Universal Robots PolyScope program: programa.urp

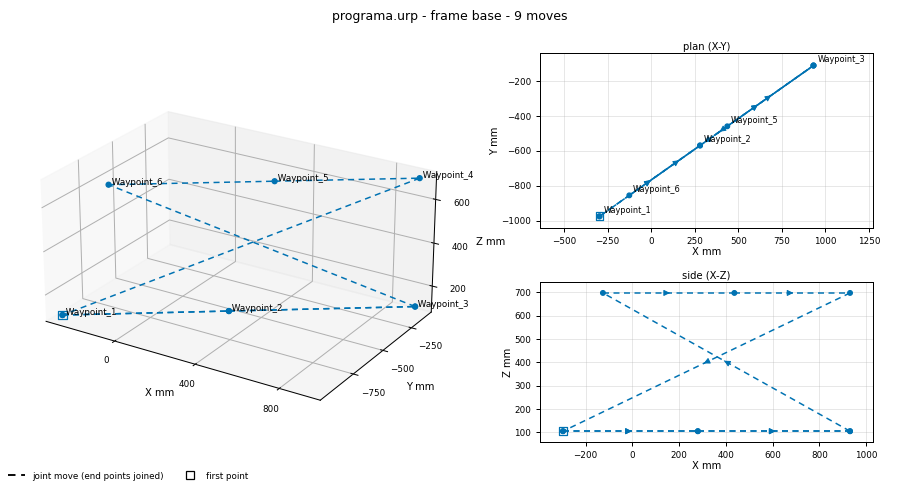
[picture p0: tool path of programa.urp in frame base, 9 of 9 moves have a stored position in this frame; points joined in program order, loops and branches not executed]
Program asdsd (installation=default directory=/home/ur/ursim-current/programs createdIn=5.8.0.10253 lastSavedIn=5.8.0.10253 robotSerialNumber=20195099999)
Calibrated DH parameters: a=[0, -0.6127, -0.57155, 0, 0, 0]; d=[0.1807, 0, 0, 0.17415, 0.11985, 0.11655]; alpha=[1.570796, 0, 0, 1.570796, -1.570796, 0]; deltaTheta=[0, 0, 0, 0, 0, 0]
InitVariablesNode variables(variable(name=cont, expression=0), variable(name=passou, expression=0))
Robot Program (runOnlyOnce=false)
  If passou≟3 (checkContinuously=true)
    Loop While (checkContinuously=false) expression=cont<6
      MoveJ speed 60 deg/s, acceleration 80 deg/s^2 (useActiveTCP=true) feature=Base
        Waypoint Waypoint_1: TCP in base x=-296.786 y=-975.284 z=105.312 mm, rx=-0.001 ry=3.1253 rz=0.0192 rad; joints [-97.186, -137.51, -82.966, -50.339, 90.834, -7.229] deg
        Waypoint Waypoint_2: TCP in base x=280.226 y=-568.577 z=105.312 mm, rx=-0.001 ry=3.1253 rz=0.0192 rad; joints [-48.039, -114.056, -131.076, -24.771, 91.162, 41.925] deg
        Waypoint Waypoint_3: TCP in base x=931.245 y=-109.705 z=105.312 mm, rx=-0.001 ry=3.1253 rz=0.0192 rad; joints [3.904, -131.88, -94.985, -42.159, 90.64, 93.872] deg
        cont := cont+1
    passou := 0
  cont := 0
  MoveJ speed 60 deg/s, acceleration 80 deg/s^2 (useActiveTCP=true) feature=Base
    Waypoint Waypoint_6: TCP in base x=-125.84 y=-854.793 z=697.554 mm, rx=-0.001 ry=3.1253 rz=0.0192 rad; joints [-86.88, -104.965, -70.738, -94.95, 90.967, 3.078] deg
    Waypoint Waypoint_5: TCP in base x=436.459 y=-458.455 z=697.554 mm, rx=-0.001 ry=3.1253 rz=0.0192 rad; joints [-30.645, -82.258, -95.201, -92.101, 91.08, 59.322] deg
    Waypoint Waypoint_4: TCP in base x=931.245 y=-109.705 z=697.554 mm, rx=-0.001 ry=3.1253 rz=0.0192 rad; joints [3.904, -112.237, -61.313, -95.475, 90.64, 93.872] deg
    Waypoint Waypoint_1: TCP in base x=-296.786 y=-975.284 z=105.312 mm, rx=-0.001 ry=3.1253 rz=0.0192 rad; joints [-97.186, -137.51, -82.966, -50.339, 90.834, -7.229] deg
    Waypoint Waypoint_2: TCP in base x=280.226 y=-568.577 z=105.312 mm, rx=-0.001 ry=3.1253 rz=0.0192 rad; joints [-48.039, -114.056, -131.076, -24.771, 91.162, 41.925] deg
    Waypoint Waypoint_3: TCP in base x=931.245 y=-109.705 z=105.312 mm, rx=-0.001 ry=3.1253 rz=0.0192 rad; joints [3.904, -131.88, -94.985, -42.159, 90.64, 93.872] deg
    passou := passou+1
